(* Schneider Machine Expert - Basic project Test_Lights, file version 3.0.0.0 *)
(* ProjectInformations: Name=Test_Lights *)

HARDWARE
  Cpu 0: TM221CE40T
  EthernetConfiguration: NetworkName=M221, IpAllocationMode=ByDhcp, IpAddress=192.168.1.10, SubnetMask=255.255.255.0
  SerialLineConfiguration: Baud=Baud19200, Parity=ParityEven, DataBits=DataBits8, StopBits=StopBits1, PhysicalMedium=PhysicalMediumRs485, TransmissionMode=TransmissionModeModbusRtu, SlaveId=1, Addressing=SlaveAddressing
  MastTask: UsePeriodScanMode=false, PeriodScan=100
  FastTask: Period=255
  CpuBehavior: StartingMode=StartAsPreviousState, AutoSaveRamOnEeprom=true, WatchdogPeriod=250

SYMBOLS  (address, symbol, comment, settings)
  %M0       SEQ_RUN  "Sequence Running"
  %TM0      TMR_LIGHT2  "Timer for Light 2"  [Mode=TON, Base=OneSecond, Preset=3]
  %TM1      TMR_LIGHT3  "Timer for Light 3"  [Mode=TON, Base=OneSecond, Preset=6]
  %I0.0     PB_START
  %I0.1     PB_STOP
  %Q0.0     LIGHT1
  %Q0.1     LIGHT2
  %Q0.2     LIGHT3

POU Test_Lights
  (* SectionNumber=1 *)

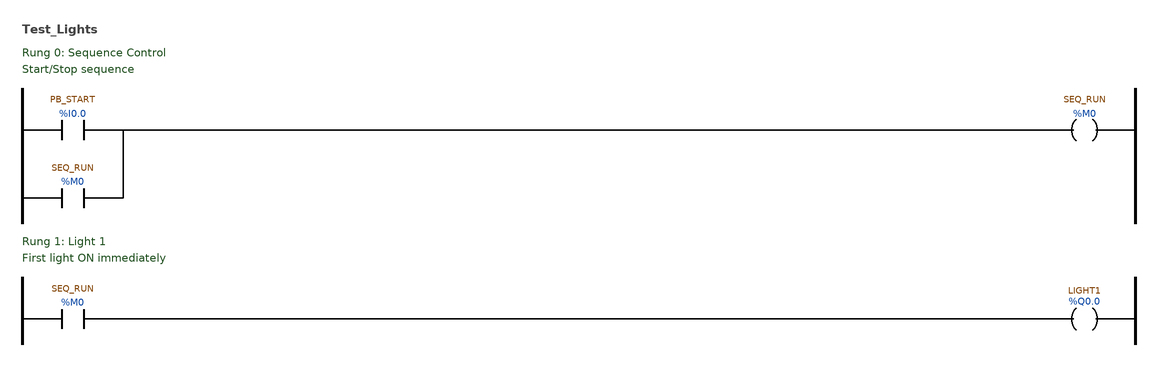

// Rung 0: Sequence Control
// Start/Stop sequence
  LD %I0.0                (* PB_START *)
  OR %M0                  (* SEQ_RUN *)
  ST %M0                  (* SEQ_RUN *)
  // as ST:
  //   SEQ_RUN := PB_START OR SEQ_RUN;

// Rung 1: Light 1
// First light ON immediately
  LD %M0                  (* SEQ_RUN *)
  ST %Q0.0                (* LIGHT1 *)
  // as ST:
  //   LIGHT1 := SEQ_RUN;
